// TwinCAT 3 PLC project ph_lv1_Communication_opcua
// Title: tclib_ph_lv1_comm_opcua
// Company: Poh
// Author: Poh
// ProjectVersion: 0.1.1.0
// ProgramVersion: 3.1.4020.1
// libraries:
//   Tc2_Standard, * (Beckhoff Automation GmbH)
//   Tc2_System, * (Beckhoff Automation GmbH)
//   Tc2_Utilities, * (Beckhoff Automation GmbH)
//   Tc3_PLCopen_OpcUa, * (Beckhoff Automation GmbH)
//   tclib_ph_lv0, * (Poh)
//   tclib_ph_lv1_generic_communication_interface, * (Poh)
// project tree:
//   Lv1_Comm_Opcua/Config/ CONFIG_OPC_SERVER.TcGVL
//   Lv1_Comm_Opcua/ C_OPC_DATACLIENT.TcPOU, C_OPC_DATASERVER.TcPOU
//   Project Information/ F_GetVersion.TcPOU
//   Version/ Global_Version.TcGVL
// (motion and I/O tree: see PLC project ph_lv0)
// real-time tasks:
//   TASK PlcTask: cycle T#10ms, priority 20, ADS port 350

// ---- Lv1_Comm_Opcua/Config/CONFIG_OPC_SERVER.TcGVL
{attribute 'qualified_only'}
VAR_GLOBAL CONSTANT
	OPC_BOOL_DATA_SIZE : INT := 10;
	OPC_SINT_DATA_SIZE : INT := 10;
	OPC_DINT_DATA_SIZE : INT := 10;
	OPC_LREAL_DATA_SIZE : INT := 10;
END_VAR

// ---- Version/Global_Version.TcGVL
{attribute 'TcGenerated'}
// This function has been automatically generated from the project information.
VAR_GLOBAL CONSTANT
	{attribute 'const_non_replaced'}
	{attribute 'linkalways'}
	stLibVersion_tclib_ph_lv1_comm_opcua : ST_LibVersion := (iMajor := 0, iMinor := 1, iBuild := 1, iRevision := 0, sVersion := '0.1.1.0');
END_VAR

// ---- Lv1_Comm_Opcua/C_OPC_DATACLIENT.TcPOU
(*
	Y:2016		M:05		D:20
	T:CLASS		N:OPC_DATACLIENT
	D:Class object for OPC UA client.
*)
FUNCTION_BLOCK C_OPC_DATACLIENT IMPLEMENTS IFC_GENERIC_COMMUNICATION_INTERFACE
VAR_INPUT
END_VAR
VAR_OUTPUT
	Message				: STRING(255);
END_VAR
VAR	
	_C_OPENCONNECTION	: UA_Connect;
	_C_CLOSECONNECTION	: UA_Disconnect;
	_C_GETNAMESPACEINDEX: UA_GetNamespaceIndex;
	_C_GETNODEHANDLE	: UA_NodeGetHandle;
	_C_RELEASENODEHANDLE: UA_NodeReleaseHandle;
	_C_READ 			: UA_Read;
	_C_WRITE 			: UA_Write;
	
	_HNDL_CONNECTION	: DWORD;
	
	_SERVER_URL				: STRING(255) := 'opc.tcp://localhost:4840';
	_ENCRYPTED_CONNECTION 	: BOOL := FALSE;
	_ENCRYPTION_128_BITS	: BOOL := FALSE;
	
	_NAMESPACE			: STRING(255);
	_NAMESPACE_INDEX	: UINT;
	_NAMESPACE_ERROR	: BOOL;
	
	_INTERNAL_STATE		: INT := 0;
	_C_GETHOSTNAME 		: FB_GetHostName;  
END_VAR

(*
	Y:2016		M:05		D:25
	D:Method to close the opened OPC UA connection in the context of a generic communication interface.
*)
METHOD Close_Connection : ph_lv0.RETURN_CODE
VAR_INPUT
END_VAR
CASE Opc_Disconnect() OF 
ph_lv0.LV0_RETURNCODE.RETURN_ERROR:
	Close_Connection := ph_lv0.LV0_RETURNCODE.RETURN_ERROR;
ph_lv0.LV0_RETURNCODE.RETURN_SUCCESS:
	Close_Connection := ph_lv0.LV0_RETURNCODE.RETURN_SUCCESS;
ELSE
	Close_Connection := ph_lv0.LV0_RETURNCODE.RETURN_BUSY;
END_CASE
END_METHOD

(*
	Y:2016		M:05		D:20
	D:Method to create the node handle in the context of a generic interface.
*)
METHOD Create_Handle : ph_lv0.RETURN_CODE
VAR_INPUT
	//.COMM_HANDLE is to be used as a STRING(255)
		Configuration	: PH_LV1_GENERIC_COMMUNICATION_INTERFACE.S_GCI_CONFIG;
	//Direct handle output
		OUT_HANDLE		: POINTER TO UDINT;
END_VAR
VAR	
	NODE_ID				: STRING(255);
	_HNDL_NODE			: DWORD;
END_VAR
MEMCPY(ADR(NODE_ID), ADR(CONFIGURATION.Comm_Handle), SIZEOF(CONFIGURATION.Comm_Handle));

CASE Get_NodeHandle(NODE_ID, ADR(_HNDL_NODE)) OF 
ph_lv0.LV0_RETURNCODE.RETURN_ERROR:
	Message := 'Unable to create handle';
	Create_Handle := ph_lv0.LV0_RETURNCODE.RETURN_ERROR;
ph_lv0.LV0_RETURNCODE.RETURN_SUCCESS:
	OUT_HANDLE^ := _HNDL_NODE;
	Create_Handle := ph_lv0.LV0_RETURNCODE.RETURN_SUCCESS;
ELSE
	Create_Handle := ph_lv0.LV0_RETURNCODE.RETURN_BUSY;
END_CASE
END_METHOD

METHOD FB_init : BOOL
VAR_INPUT
	bInitRetains : BOOL; // if TRUE, the retain variables are initialized (warm start / cold start)
	bInCopyCode : BOOL;  // if TRUE, the instance afterwards gets moved into the copy code (online change)
	ENCRYPTED_CONNECTION 	: BOOL := FALSE;
	ENCRYPTION_128_BITS		: BOOL := FALSE;
	SERVER_URL 				: STRING(255);
	OPC_NAMESPACE 				: STRING(255);
END_VAR
_ENCRYPTED_CONNECTION 	:= ENCRYPTED_CONNECTION;
_ENCRYPTION_128_BITS	:= ENCRYPTION_128_BITS;
_SERVER_URL := SERVER_URL;
_NAMESPACE := OPC_NAMESPACE;
END_METHOD

(*
	Y:2016		M:05		D:20
	D:Not recommended for use. Method to reset the internal connection details even if the base function fails.
*)
METHOD Force_Close_Connection : ph_lv0.RETURN_CODE
VAR_INPUT
END_VAR
_C_CLOSECONNECTION(
	Execute:= TRUE, 
	ConnectionHdl:= _HNDL_CONNECTION);
IF _C_CLOSECONNECTION.Error THEN
	_C_CLOSECONNECTION(
		Execute:= FALSE );
	//CLEAN UP
		_HNDL_CONNECTION := 0;
		_NAMESPACE_INDEX := 0;
		MEMSET(ADR(_NAMESPACE), 0, SIZEOF(_NAMESPACE));
	Force_Close_Connection := ph_lv0.LV0_RETURNCODE.RETURN_SUCCESS - 1;
ELSIF _C_CLOSECONNECTION.Done AND NOT _C_CLOSECONNECTION.Busy THEN
	_C_CLOSECONNECTION(
		Execute:= FALSE );
	//CLEAN UP
		_HNDL_CONNECTION := 0;
		_NAMESPACE_INDEX := 0;
		MEMSET(ADR(_NAMESPACE), 0, SIZEOF(_NAMESPACE));
	Force_Close_Connection := ph_lv0.LV0_RETURNCODE.RETURN_SUCCESS;
ELSE
	Force_Close_Connection := ph_lv0.LV0_RETURNCODE.RETURN_BUSY;
END_IF
END_METHOD

(*
	Y:2016		M:05		D:20
	D:Method for getting the host-name of the target AMS device. Works for TCP-IP based connections.
*)
METHOD Get_HostName : RETURN_CODE
VAR_INPUT
	TARGET_DEVICE	: T_AmsNetId;
	REF_OUT			: POINTER TO STRING(255);
END_VAR
VAR
	_BUFFER 		: STRING(255);
END_VAR
_C_GETHOSTNAME(
	sNetID:= TARGET_DEVICE, 
	bExecute:= TRUE,
	sHostName=> _BUFFER);
IF _C_GETHOSTNAME.bError THEN
	_C_GETHOSTNAME(
		bExecute:= FALSE);
	Get_HostName := ph_lv0.LV0_RETURNCODE.RETURN_ERROR;
ELSIF NOT _C_GETHOSTNAME.bBusy AND NOT _C_GETHOSTNAME.bError THEN
	_C_GETHOSTNAME(
		bExecute:= FALSE);
	MEMSET(REF_OUT, 0, SIZEOF(REF_OUT^));
	MEMCPY(REF_OUT, ADR(_BUFFER), LEN(_BUFFER));
	Get_HostName := ph_lv0.LV0_RETURNCODE.RETURN_SUCCESS;
ELSE
	Get_HostName := ph_lv0.LV0_RETURNCODE.RETURN_BUSY;
END_IF
END_METHOD

(*
	Y:2016		M:05		D:20
	D:Method to obtain the node handle. Supports string identifier only.
*)
METHOD Get_NodeHandle : ph_lv0.RETURN_CODE
VAR_INPUT
	NODE_ID				: STRING(255);
	NODE_HANDLE			: POINTER TO DWORD;
END_VAR
VAR	
	_STNodeInfo			: ST_UANodeId;
	_HNDL_NODE			: DWORD;
END_VAR
_STNodeInfo.eIdentifierType := E_UAIdentifierType.eUAIdentifierType_String;
_STNodeInfo.nNamespaceIndex := _NAMESPACE_INDEX;

_STNodeInfo.sIdentifier := NODE_ID;

_C_GETNODEHANDLE(
	Execute:= TRUE, 
	ConnectionHdl:= _HNDL_CONNECTION, 
	NodeID:= _STNodeInfo, 
	NodeHdl=> _HNDL_NODE );
IF _C_GETNODEHANDLE.Error THEN
	_C_GETNODEHANDLE(
		Execute:= FALSE );		
	Get_NodeHandle := ph_lv0.LV0_RETURNCODE.RETURN_ERROR;
ELSIF _C_GETNODEHANDLE.Done AND NOT _C_GETNODEHANDLE.Busy THEN
	MEMCPY(NODE_HANDLE, ADR(_HNDL_NODE), SIZEOF(_HNDL_NODE));
	_C_GETNODEHANDLE(
		Execute:= FALSE );
	Get_NodeHandle := ph_lv0.LV0_RETURNCODE.RETURN_SUCCESS;
ELSE
	Get_NodeHandle := ph_lv0.LV0_RETURNCODE.RETURN_BUSY;
END_IF
END_METHOD

PROPERTY Namespace : STRING(255)
GET
Namespace := _NAMESPACE;
END_GET
END_PROPERTY

PROPERTY Namespace_Index : UINT
GET
Namespace_Index := _NAMESPACE_INDEX;
END_GET
END_PROPERTY

METHOD PRIVATE Opc_Connect : ph_lv0.RETURN_CODE
VAR_INPUT
END_VAR
VAR	
	_STConnectionInfo	: ST_UASessionConnectInfo; 
END_VAR
IF _ENCRYPTED_CONNECTION THEN
	_STConnectionInfo.eSecurityMode := E_UASecurityMsgMode.eUASecurityMsgMode_Sign_Encrypt;
ELSE
	_STConnectionInfo.eSecurityMode := E_UASecurityMsgMode.eUASecurityMsgMode_None;
END_IF

IF NOT _ENCRYPTED_CONNECTION THEN
	_STConnectionInfo.eSecurityPolicyUri := E_UASecurityPolicy.eUASecurityPolicy_None; 
ELSIF _ENCRYPTION_128_BITS THEN
	_STConnectionInfo.eSecurityPolicyUri := E_UASecurityPolicy.eUASecurityPolicy_Basic128Rsa15; 
ELSE
	_STConnectionInfo.eSecurityPolicyUri := E_UASecurityPolicy.eUASecurityPolicy_Basic256; 
END_IF

_STConnectionInfo.eTransportProfileUri 	:= E_UATransportProfile.eUATransportProfileUri_UATcp;
_STConnectionInfo.tConnectTimeout 		:= T#30S;
_STConnectionInfo.tSessionTimeout 		:= T#30S;

_C_OPENCONNECTION(
	Execute:= TRUE, 
	ServerUrl:= _SERVER_URL, 
	SessionConnectInfo:= _stConnectionInfo, 
	Timeout:= , 
	ConnectionHdl=> _HNDL_CONNECTION );

IF _C_OPENCONNECTION.Error THEN
	_C_OPENCONNECTION(
		Execute:= FALSE );
	Opc_Connect := ph_lv0.LV0_RETURNCODE.RETURN_ERROR;
ELSIF _C_OPENCONNECTION.Done AND NOT _C_OPENCONNECTION.Busy THEN
	_C_OPENCONNECTION(
		Execute:= FALSE );
	Opc_Connect := ph_lv0.LV0_RETURNCODE.RETURN_SUCCESS;
ELSE
	Opc_Connect := ph_lv0.LV0_RETURNCODE.RETURN_BUSY;
END_IF
END_METHOD

(*
	Y:2016		M:05		D:25
	D:Method to close the opened OPC UA connection
*)
METHOD PRIVATE Opc_Disconnect : RETURN_CODE
VAR_INPUT
END_VAR
VAR	
END_VAR
IF _HNDL_CONNECTION <> 0 THEN	
	_C_CLOSECONNECTION(
		Execute:= TRUE, 
		ConnectionHdl:= _HNDL_CONNECTION);
	IF _C_CLOSECONNECTION.Error THEN
		_C_CLOSECONNECTION(
			Execute:= FALSE );
		Opc_Disconnect := ph_lv0.LV0_RETURNCODE.RETURN_ERROR;
	ELSIF _C_CLOSECONNECTION.Done AND NOT _C_CLOSECONNECTION.Busy THEN
		_C_CLOSECONNECTION(
			Execute:= FALSE );
		//CLEAN UP
			_HNDL_CONNECTION := 0;
			_NAMESPACE_INDEX := 0;
			MEMSET(ADR(_NAMESPACE), 0, SIZEOF(_NAMESPACE));
		Opc_Disconnect := ph_lv0.LV0_RETURNCODE.RETURN_SUCCESS;
	ELSE
		Opc_Disconnect := ph_lv0.LV0_RETURNCODE.RETURN_BUSY;
	END_IF
ELSE
	Opc_Disconnect := ph_lv0.LV0_RETURNCODE.RETURN_SUCCESS;
END_IF
END_METHOD

METHOD PRIVATE Opc_Read : ph_lv0.RETURN_CODE
VAR_INPUT
	NODE_HANDLE	: DWORD;
	DATA		: PVOID;
	DATA_SIZE 	: UDINT;
	OPCUA_START_INDEX 	: UDINT;
	OPCUA_END_INDEX		: UDINT;
END_VAR
VAR	
	_STNodeAddInfo		: ST_UANodeAdditionalInfo;
	_STNodeIndexRange	: ST_UAIndexRange;
END_VAR
_STNodeIndexRange.nStartIndex := OPCUA_START_INDEX;
_STNodeIndexRange.nEndIndex := OPCUA_END_INDEX;

_STNodeAddInfo.nIndexRangeCount := 1;
_STNodeAddInfo.stIndexRange[1] := _STNodeIndexRange;

_C_READ(
	Execute:= TRUE, 
	ConnectionHdl:= _HNDL_CONNECTION, 
	NodeHdl:= NODE_HANDLE, 
	stNodeAddInfo:= _STNodeAddInfo, 
	pVariable:= DATA, 
	cbData:= DATA_SIZE );
	
IF _C_READ.Error THEN
	_C_READ(
		Execute:= FALSE );
	Opc_Read := ph_lv0.LV0_RETURNCODE.RETURN_ERROR;
ELSIF _C_READ.Done AND NOT _C_READ.Busy THEN
	_C_READ(
		Execute:= FALSE );
	Opc_Read := ph_lv0.LV0_RETURNCODE.RETURN_SUCCESS;
ELSE
	Opc_Read := ph_lv0.LV0_RETURNCODE.RETURN_BUSY;
END_IF
END_METHOD

METHOD PRIVATE Opc_Write : ph_lv0.RETURN_CODE
VAR_INPUT
	NODE_HANDLE			: DWORD;
	DATA				: PVOID;
	DATA_SIZE 			: UDINT;
	OPCUA_START_INDEX 	: UDINT;
	OPCUA_END_INDEX		: UDINT;
END_VAR
VAR	
	_STNodeAddInfo		: ST_UANodeAdditionalInfo;
	_STNodeIndexRange	: ST_UAIndexRange;
END_VAR
_STNodeIndexRange.nStartIndex := OPCUA_START_INDEX;
_STNodeIndexRange.nEndIndex := OPCUA_END_INDEX;

_STNodeAddInfo.nIndexRangeCount := 1;
_STNodeAddInfo.stIndexRange[1] := _STNodeIndexRange;

_C_WRITE(
	Execute:= TRUE, 
	ConnectionHdl:= _HNDL_CONNECTION, 
	NodeHdl:= NODE_HANDLE, 
	stNodeAddInfo:= , 
	pVariable:= DATA, 
	cbData:= DATA_SIZE );
IF _C_WRITE.Error THEN
	_C_WRITE(
		Execute:= FALSE );
	Opc_Write := ph_lv0.LV0_RETURNCODE.RETURN_ERROR;
ELSIF _C_WRITE.Done AND NOT _C_WRITE.Busy THEN
	_C_WRITE(
		Execute:= FALSE );
	Opc_Write := ph_lv0.LV0_RETURNCODE.RETURN_SUCCESS;
ELSE
	Opc_Write := ph_lv0.LV0_RETURNCODE.RETURN_BUSY;
END_IF
END_METHOD

(*
	Y:2016		M:05		D:20
	D:Method to open the OPC UA connection.
*)
METHOD Open_Connection : ph_lv0.RETURN_CODE
VAR_INPUT
	CONNECTION_INFO : S_GCI_CONFIG;
END_VAR
VAR	
	_STConnectionInfo	: ST_UASessionConnectInfo; 
	_Status : INT := 0;
END_VAR
CASE _INTERNAL_STATE OF 
-1:
	_Status := 1;
0:
	IF _HNDL_CONNECTION <> 0 THEN
		//CONNECTION EXISTS, THEREFORE GO TO OPC UA NAMESPACE RESOLUTION
			_INTERNAL_STATE := 2;		
	ELSE
		//NO EXISTING CONNECTION, THEREFORE OPENS INITIAL CONNECTION
			_INTERNAL_STATE := 1;		
	END_IF
1:
	CASE Opc_Connect() OF 
	ph_lv0.LV0_RETURNCODE.RETURN_SUCCESS:
			MEMSET(ADR(_NAMESPACE), 0, SIZEOF(_NAMESPACE));
		_INTERNAL_STATE := _INTERNAL_STATE + 1;
	ph_lv0.LV0_RETURNCODE.RETURN_ERROR:
		Message := 'Unable to open OPC UA connection';
		_INTERNAL_STATE := 1;
	END_CASE
2:
	MEMCPY(ADR(CONNECTION_INFO.Comm_Handle), ADR(_NAMESPACE), SIZEOF(CONNECTION_INFO.Comm_Handle));
	CASE Set_Namespace(_NAMESPACE) OF
	ph_lv0.LV0_RETURNCODE.RETURN_SUCCESS:
		_INTERNAL_STATE := _INTERNAL_STATE + 1;
	ph_lv0.LV0_RETURNCODE.RETURN_ERROR:
		Message := 'Unable to find OPC UA namespace';
		_INTERNAL_STATE := 1;
	END_CASE
3:
	_Status := -1;
END_CASE

//Method return
	CASE _Status OF 
		-1:
			_INTERNAL_STATE := 0;
			MEMSET(ADR(Message), 0, SIZEOF(Message));
			Open_Connection := ph_lv0.LV0_RETURNCODE.RETURN_SUCCESS;
		1:
			_INTERNAL_STATE := 0;
			Open_Connection := ph_lv0.LV0_RETURNCODE.RETURN_ERROR;
		ELSE
			Open_Connection := ph_lv0.LV0_RETURNCODE.RETURN_BUSY;
	END_CASE
END_METHOD

(*
	Y:2016		M:05		D:20
	D:Method for opc ua read in the context of a generic interface.
*)
METHOD Read : RETURN_CODE
VAR_INPUT
	Configuration	: S_GCI_CONFIG;
END_VAR
VAR	
	NODE_HANDLE			: DWORD;
	DATA				: PVOID;
	DATA_SIZE 			: UDINT;
	OPCUA_START_INDEX 	: UDINT;
	OPCUA_END_INDEX		: UDINT;
	_STNodeAddInfo		: ST_UANodeAdditionalInfo;
	_STNodeIndexRange	: ST_UAIndexRange;
END_VAR
_STNodeIndexRange.nStartIndex := OPCUA_START_INDEX;
_STNodeIndexRange.nEndIndex := OPCUA_END_INDEX;

_STNodeAddInfo.nIndexRangeCount := 1;
_STNodeAddInfo.stIndexRange[1] := _STNodeIndexRange;

_C_READ(
	Execute:= TRUE, 
	ConnectionHdl:= _HNDL_CONNECTION, 
	NodeHdl:= NODE_HANDLE, 
	stNodeAddInfo:= _STNodeAddInfo, 
	pVariable:= DATA, 
	cbData:= DATA_SIZE );
	
IF _C_READ.Error THEN
	_C_READ(
		Execute:= FALSE );
	Read := ph_lv0.LV0_RETURNCODE.RETURN_ERROR;
ELSIF _C_READ.Done AND NOT _C_READ.Busy THEN
	_C_READ(
		Execute:= FALSE );
	Read := ph_lv0.LV0_RETURNCODE.RETURN_SUCCESS;
ELSE
	Read := ph_lv0.LV0_RETURNCODE.RETURN_BUSY;
END_IF
END_METHOD

(*
	Y:2016		M:05		D:20
	D:Method to release the node handle in the context of a generic interface.
*)
METHOD Release_Handle : RETURN_CODE
VAR_INPUT
	//Direct handle input.
		IN_HANDLE	: POINTER TO UDINT;
END_VAR
CASE Release_NodeHandle(IN_HANDLE^) OF 
ph_lv0.LV0_RETURNCODE.RETURN_ERROR:
	Message := 'Unable to release handle';
	Release_Handle := ph_lv0.LV0_RETURNCODE.RETURN_ERROR;
ph_lv0.LV0_RETURNCODE.RETURN_SUCCESS:
	IN_HANDLE^ := 0;
	Release_Handle := ph_lv0.LV0_RETURNCODE.RETURN_SUCCESS;
ELSE
	Release_Handle := ph_lv0.LV0_RETURNCODE.RETURN_BUSY;	
END_CASE
END_METHOD

METHOD PRIVATE Release_NodeHandle : RETURN_CODE
VAR_INPUT
	NODE_HANDLE : DWORD;
END_VAR
_C_RELEASENODEHANDLE(
	Execute:= TRUE, 
	ConnectionHdl:= _HNDL_CONNECTION, 
	NodeHdl:= NODE_HANDLE );
IF _C_RELEASENODEHANDLE.Error THEN
	_C_RELEASENODEHANDLE(
		Execute:= FALSE );		
	Release_NodeHandle := ph_lv0.LV0_RETURNCODE.RETURN_ERROR;
ELSIF _C_RELEASENODEHANDLE.Done AND NOT _C_RELEASENODEHANDLE.Busy THEN
	_C_RELEASENODEHANDLE(
		Execute:= FALSE );
	Release_NodeHandle := ph_lv0.LV0_RETURNCODE.RETURN_SUCCESS;
ELSE
	Release_NodeHandle := ph_lv0.LV0_RETURNCODE.RETURN_BUSY;
END_IF
END_METHOD

PROPERTY Server_Url : STRING(255)
GET
Server_Url := _SERVER_URL;
END_GET
END_PROPERTY

(*
	Y:2016		M:05		D:20
	D:Method to configure the OPC UA server namespace.
*)
METHOD Set_Namespace : RETURN_CODE
VAR_INPUT
	//The namespace of the variables in the OPC UA. Eg. 'urn:HOST-NAME:BeckhoffAutomation:Ua:PLC1' 
		Namespace : STRING(255);
END_VAR
_C_GETNAMESPACEINDEX(
	Execute:= TRUE, 
	ConnectionHdl:= _HNDL_CONNECTION, 
	NamespaceUri:= Namespace );
IF _C_GETNAMESPACEINDEX.Error THEN
	_C_GETNAMESPACEINDEX(
	Execute:= FALSE );
	Set_Namespace := ph_lv0.LV0_RETURNCODE.RETURN_ERROR;
ELSIF _C_GETNAMESPACEINDEX.Done AND NOT _C_GETNAMESPACEINDEX.Busy THEN
	_NAMESPACE 			:= Namespace;
	_NAMESPACE_INDEX 	:= _C_GETNAMESPACEINDEX.NamespaceIndex;
	_C_GETNAMESPACEINDEX(
		Execute:= FALSE );
	Set_Namespace := ph_lv0.LV0_RETURNCODE.RETURN_SUCCESS;
ELSE
	Set_Namespace := ph_lv0.LV0_RETURNCODE.RETURN_BUSY;
END_IF
END_METHOD

(*
	Y:2016		M:05		D:20
	D:Method to configure the OPC UA connection's security policy.
*)
METHOD Set_Security_Config : RETURN_CODE
VAR_INPUT
	//Determines if the connection is signed and encrypted.
		ENCRYPTED_CONNECTION 	: BOOL := FALSE;
	//Determines the encryption length of the connection. 128-bits/254-bits.
		ENCRYPTION_128_BITS	: BOOL := FALSE;
END_VAR
IF _HNDL_CONNECTION <> 0 THEN
	Message := 'Close connection before changing the connection$'s security settings';
	Set_Security_Config := ph_lv0.LV0_RETURNCODE.RETURN_ERROR;
ELSE
	_ENCRYPTED_CONNECTION := ENCRYPTED_CONNECTION;
	_ENCRYPTION_128_BITS := ENCRYPTION_128_BITS;
	Set_Security_Config := ph_lv0.LV0_RETURNCODE.RETURN_SUCCESS;
END_IF
END_METHOD

(*
	Y:2016		M:05		D:20
	D:Method to configure the server URL for the OPC UA connection.
*)
METHOD Set_Server_Url : RETURN_CODE
VAR_INPUT
	//The OPC UA server's url. Eg. opc.tcp://host-name:4840
		Url : STRING(255);
END_VAR
IF _HNDL_CONNECTION <> 0 THEN
	Message := 'Close connection before changing the server URL';
	Set_Server_Url := ph_lv0.LV0_RETURNCODE.RETURN_ERROR;
ELSE
	_SERVER_URL := URL;
	Set_Server_Url := ph_lv0.LV0_RETURNCODE.RETURN_SUCCESS;
END_IF
END_METHOD

METHOD Write : RETURN_CODE
VAR_INPUT
	Configuration	: S_GCI_CONFIG;
END_VAR
VAR	
	NODE_HANDLE			: DWORD;
	DATA				: PVOID;
	DATA_SIZE 			: UDINT;
	OPCUA_START_INDEX 	: UDINT;
	OPCUA_END_INDEX		: UDINT;
	_STNodeAddInfo		: ST_UANodeAdditionalInfo;
	_STNodeIndexRange	: ST_UAIndexRange;
END_VAR
_STNodeIndexRange.nStartIndex := OPCUA_START_INDEX;
_STNodeIndexRange.nEndIndex := OPCUA_END_INDEX;

_STNodeAddInfo.nIndexRangeCount := 1;
_STNodeAddInfo.stIndexRange[1] := _STNodeIndexRange;

_C_WRITE(
	Execute:= TRUE, 
	ConnectionHdl:= _HNDL_CONNECTION, 
	NodeHdl:= NODE_HANDLE, 
	stNodeAddInfo:= , 
	pVariable:= DATA, 
	cbData:= DATA_SIZE );
IF _C_WRITE.Error THEN
	_C_WRITE(
		Execute:= FALSE );
	Write := ph_lv0.LV0_RETURNCODE.RETURN_ERROR;
ELSIF _C_WRITE.Done AND NOT _C_WRITE.Busy THEN
	_C_WRITE(
		Execute:= FALSE );
	Write := ph_lv0.LV0_RETURNCODE.RETURN_SUCCESS;
ELSE
	Write := ph_lv0.LV0_RETURNCODE.RETURN_BUSY;
END_IF
END_METHOD

END_FUNCTION_BLOCK

// ---- Lv1_Comm_Opcua/C_OPC_DATASERVER.TcPOU
FUNCTION_BLOCK C_OPC_DATASERVER
VAR_INPUT
END_VAR
VAR_OUTPUT
END_VAR
VAR
	{attribute 'OPC.UA.DA' := '1'}
	DATA_BOOL : ARRAY[0..CONFIG_OPC_SERVER.OPC_BOOL_DATA_SIZE] OF BOOL;
	{attribute 'OPC.UA.DA' := '1'}
	DATA_SINT : ARRAY[0..CONFIG_OPC_SERVER.OPC_SINT_DATA_SIZE] OF SINT;
	{attribute 'OPC.UA.DA' := '1'}
	DATA_DINT : ARRAY[0..CONFIG_OPC_SERVER.OPC_DINT_DATA_SIZE] OF DINT;
	{attribute 'OPC.UA.DA' := '1'}
	DATA_LREAL : ARRAY[0..CONFIG_OPC_SERVER.OPC_LREAL_DATA_SIZE] OF LREAL;	
END_VAR

END_FUNCTION_BLOCK

// ---- Project Information/F_GetVersion.TcPOU
// This function has been automatically generated from the project information.
{attribute 'signature_flag' := '1073741824'}
{attribute 'TcGenerated'}
FUNCTION F_GetVersion : ST_LibVersion
VAR_INPUT
	
END_VAR

F_GetVersion.iMajor := 0;
F_GetVersion.iMinor := 1;
F_GetVersion.iBuild := 1;
F_GetVersion.iRevision := 0;

END_FUNCTION
